(* CODESYS project 07052026.export

Project tree, tasks and I/O mapping:
  Device : ctrlX CORE ARM64, Bosch Rexroth AG, version 3.6.3.0
    application Application
      libraries: CXA_Datalayer, * (Bosch Rexroth AG); CXA_FileAsync, * (Bosch Rexroth AG); CXA_Motion, * (Bosch Rexroth AG); CXA_PLCopen, * (Bosch Rexroth AG); CXA_RobotFastManagement, 3.6.2.1 (Bosch Rexroth spa); VisuDialogs, * (System); CXA_EthercatMaster, * (Bosch Rexroth AG)
      task MainTask (cyclic, interval t#20ms, priority 30) calls PLC_PRG, prgRobotManagement, POU_GetBusState
      Robot_management_AddsOn/
        data type HomeStruct
        _CXA_RobotFastManagement_3_6_1_5/
          _00_RobotCofigurationSettings/
            global variables GVL_Robot_Config_Settings
          _01_GlobalVarConstRobotBase_3_6_1_5/
            global variables Global_Var_RobotBase
          _02_GlobalVarConstantRobotPathPlanner_3_6_1_5/
            global variables Global_Var_RobotPathPlanner
          _05_GlobalBeltVar_1_0/
            global variables GlobalBeltVar
          _06_RobotProgramExample_3_6_1_5/
            program prgRobotManagement [ST]: a00_RobotBase, a01_PathPlanner, a02_TeachIn, a03_Belt, a99_Examples
      global variables GVL
      program PLC_PRG [ST]
      program POU_GetBusState [ST]
      data type DUT
      trace Delta (task MainTask): stRobotFbk[1].arPathCoordinates[1], stRobotFbk[1].arPathCoordinates[2], stRobotFbk[1].arPathCoordinates[3], stRobotFbk[1].rPathVelocity, stRobotFbk[1].rPathAcceleration, stRobotFbk[1].rPathJerk, stKinPathBlendingStatus[1].bKinContourActive, stKinPathBlendingStatus[1].bPolySlopeActive, PLC_PRG.bCycleStart, stRobotPathPlanner[1].stRobotPoints[2].bMoveToDone, prgRobotManagement.fbRobotPathPlanner[1].fbMoveAbsolute1.I_SetPointType, prgRobotManagement.fbRobotPathPlanner[1].fbMoveAbsolute1.O_bKinMoveLinAbsError, PLC_PRG.bSetDriveOutput, prgRobotManagement.fbRobotPathPlanner[1].O_stPathPlannerFbk.usiBufferedBlock, prgRobotManagement.fbRobotPathPlanner[1].i, prgRobotManagement.fbRobotPathPlanner[1].bExMove, prgRobotManagement.fbRobotPathPlanner[1].iStep, prgRobotManagement.fbRobotPathPlanner[1].iBufferValue, prgRobotManagement.fbRobotPathPlanner[1].iBufferLimit, , prgRobotManagement.fbRobotPathPlanner[1].iCountCmdBuffered, PLC_PRG.fbIpoDelta.Position[1], PLC_PRG.fbIpoDelta.Position[2], PLC_PRG.fbIpoDelta.Position[3], prgRobotManagement.tCycle, PLC_PRG.bEnableCiclo, PLC_PRG.rRot, PLC_PRG.rRadius
      trace Scara (task MainTask): stRobotFbk[2].arPathCoordinates[1], stRobotFbk[2].arPathCoordinates[2], stRobotFbk[2].arPathCoordinates[6], stRobotFbk[2].rPathVelocity, stRobotFbk[2].rPathAcceleration, stRobotFbk[2].rPathJerk, stKinPathBlendingStatus[2].bKinContourActive, stKinPathBlendingStatus[2].bPolySlopeActive, PLC_PRG.bCycleStart, stRobotPathPlanner[1].stRobotPoints[2].bMoveToDone, prgRobotManagement.fbRobotPathPlanner[2].fbMoveAbsolute1.I_SetPointType, prgRobotManagement.fbRobotPathPlanner[2].fbMoveAbsolute1.O_bKinMoveLinAbsError, PLC_PRG.bSetDriveOutput, prgRobotManagement.fbRobotPathPlanner[2].O_stPathPlannerFbk.usiBufferedBlock, prgRobotManagement.fbRobotPathPlanner[2].i, prgRobotManagement.fbRobotPathPlanner[2].bExMove, prgRobotManagement.fbRobotPathPlanner[2].iStep, prgRobotManagement.fbRobotPathPlanner[2].iBufferValue, prgRobotManagement.fbRobotPathPlanner[1].iBufferLimit, , prgRobotManagement.fbRobotPathPlanner[2].iCountCmdBuffered, PLC_PRG.fbIpoDelta.Position[1], PLC_PRG.fbIpoDelta.Position[2], PLC_PRG.fbIpoDelta.Position[3], prgRobotManagement.tCycle, PLC_PRG.bEnableCiclo, PLC_PRG.rRot, PLC_PRG.rRadius
      visualisation Visualization
    Realtime_Data : DataLayer, Bosch Rexroth AG, version 3.6.2.0
  text list GlobalTextList
*)

// Device/Application/DUT
{attribute 'qualified_only'}
{attribute 'strict'}
TYPE DUT :
(
	enum_member := 0
);
END_TYPE

// Device/Application/Robot_management_AddsOn/HomeStruct
TYPE HomeStruct :
STRUCT
    FsSdoSetUp_u : UINT;
	SlaveAddress : UINT;
	WorkingMode : UINT;
    FsHoming : UINT;
    OuterAngle : REAL;
	OffesetInnerAngle_w : DINT;
	OffesetInnerAngle_r : DINT;
	HomeOffsetDone : BOOL;
	FeedConstant_w : ULINT;
	GearRatio_sub1_w : ULINT;
	GearRatio_sub2_w : ULINT;
	FeedConstant_r : ULINT;
	GearRatio_sub1_r : ULINT;
	GearRatio_sub2_r : ULINT;
	GearRatioConstant : REAL;
END_STRUCT
END_TYPE

// Device/Application/GVL
//{attribute 'qualified_only'}

VAR_GLOBAL
	//st values
	IN_OP_NO_HOMING   : UINT   			   := 0;
	FROM_OP_PREOP_HOME_NOT_DONE   : UINT   := 1;
	HOMING_DONE   : UINT   				   := 2;
	FROM_PREOP_OP_HOME_DONE   : UINT       := 3;

	HOMING_MODE : UINT := 0;
	FEED_CONSTANT : UINT := 1;
	GEAR_RATIO_SUB1 : UINT := 2;
	GEAR_RATIO_SUB2 : UINT := 3;
	METH_AND_ANGLE : UINT := 4;
	WRITE_OFFSET : UINT := 5;

	re_offset_input_angle : REAL := 0;
	ArrayCounter : UINT := 0;
	
    ElacArrayHoming : ARRAY[0..1] OF HomeStruct := [
        (
            FsSdoSetUp_u := 0,
            SlaveAddress := 1001,
			WorkingMode := 0, 
            FsHoming := 0,
            OuterAngle := 700000,
            OffesetInnerAngle_w := 700000,
			OffesetInnerAngle_r := 0,
			HomeOffsetDone := FALSE,
			FeedConstant_w := 7000,
			GearRatio_sub1_w := 1,
			GearRatio_sub2_w := 1,
			FeedConstant_r := 0,
			GearRatio_sub1_r := 0,
			GearRatio_sub2_r := 0,
			GearRatioConstant := -100
        ),
        (
            FsSdoSetUp_u := 0,
            SlaveAddress := 1002,
			WorkingMode := 0, 
            FsHoming := 0,
            OuterAngle := 700000,
            OffesetInnerAngle_w := 700000,
			OffesetInnerAngle_r := 0,
			HomeOffsetDone := FALSE,
			FeedConstant_w := 7000,
			GearRatio_sub1_w := 1,
			GearRatio_sub2_w := 1,
			FeedConstant_r := 0,
			GearRatio_sub1_r := 0,
			GearRatio_sub2_r := 0,
			GearRatioConstant := -100
        )
    ];

END_VAR

// Device/Application/Robot_management_AddsOn/_CXA_RobotFastManagement_3_6_1_5/_00_RobotCofigurationSettings/GVL_Robot_Config_Settings
	///#############################################################################################
	///  #############################################################################################
	///
	///   General Header
	///  ---------------------------------------------------------------------------------------------
	///   Shortdescription       :  
	///   Version                : 1.0.0.<br>
	///   Name                   : GT DCIT/STS<br>
	///   Date                   : 2024-10-25<br>
	///   Company                : Bosch Rexroth  S.p.A. Electric Drives and Controls<br>
	///   Target                 : CtrlX Core V.2.6.4 <br>
	///   Functional description : Define here the robots and robots Axis names
	///   Handling specials      : 
	///								* global var arRobotKinConfig name must not be changed.
	///							    * axis definition global var arRobot..n..AxisConfig name could be changed
	///								  but thenew name must be update in global var arRobotKinConfig too. 									
	///	
	///								
	///  ---------------------------------------------------------------------------------------------
	///
	///   Additional Header
	///  ---------------------------------------------------------------------------------------------
	///   Used global variables  : 
	///
	///   Used Standard Library  : []	
	///
	///   Used Standard Function Block:	
	///      
	///   Possible error codes:	
	///
	///   Last Modified Issues: 
	///											
	///  -----------------------------------------------------------------------
	///
	///
	///  ---------------------------------------------------------------------------------------------
	///
	///  #############################################################################################
	///  ############################################################################################# 
VAR_GLOBAL
	arRobot1AxisConfig: ARRAY[1..16] OF ST_AXIS_REF := [(AxisRef := (AxisName := 'Axis_1'), AxisNo := 1, AxisConfig := enPositioningAxis, AxisType := enVirtualAxis), 
														(AxisRef := (AxisName := 'Axis_2'), AxisNo := 2, AxisConfig := enPositioningAxis, AxisType := enVirtualAxis), 
														(AxisRef := (AxisName := 'Axis_3'), AxisNo := 3, AxisConfig := enPositioningAxis, AxisType := enVirtualAxis),
														(AxisRef := (AxisName := 'Axis_4'), AxisNo := 4, AxisConfig := enPositioningAxis, AxisType := enVirtualAxis), 
														(AxisRef := (AxisName := 'Axis_5'), AxisNo := 5, AxisConfig := enPositioningAxis, AxisType := enVirtualAxis), 
														(AxisRef := (AxisName := 'Axis_6'), AxisNo := 6, AxisConfig := enPositioningAxis, AxisType := enVirtualAxis)];
														
														
	arRobotKinConfig: ARRAY[1..16] OF ST_KIN_REF := [	(KinRef := (KinName := 'Rob_Arm_5dof'), KinNo := 1, arAxisRef := arRobot1AxisConfig )];
END_VAR

// Device/Application/Robot_management_AddsOn/_CXA_RobotFastManagement_3_6_1_5/_01_GlobalVarConstRobotBase_3_6_1_5/Global_Var_RobotBase
{attribute 'symbol' := 'readwrite'}
{attribute 'linkalways' := ''}
VAR_GLOBAL
	///#############################################################################################
	///  #############################################################################################
	///
	///   General Header
	///  ---------------------------------------------------------------------------------------------
	///   Shortdescription       :  
	///   Version                : 1.0.0.<br>
	///   Name                   : GT DCIT/STS<br>
	///   Date                   : 2024-10-25<br>
	///   Company                : Bosch Rexroth  S.p.A. Electric Drives and Controls<br>
	///   Target                 : CtrlX Core V.2.6.4 <br>
	///   Functional description :  
	///   Handling specials      : 
	///							
	///	
	///								
	///  ---------------------------------------------------------------------------------------------
	///
	///   Additional Header
	///  ---------------------------------------------------------------------------------------------
	///   Used global variables  : 
	///
	///   Used Standard Library  : []	
	///
	///   Used Standard Function Block:	
	///      
	///   Possible error codes:	
	///
	///   Last Modified Issues: 
	///											
	///  -----------------------------------------------------------------------
	///
	///
	///  ---------------------------------------------------------------------------------------------
	///
	///  #############################################################################################
	///  ############################################################################################# 
	stRobotCmd: ARRAY[1..C_usiRobotNo] OF ST_Robot_CMD;
	stRobotFbk: ARRAY[1..C_usiRobotNo] OF ST_Robot_FBK;
END_VAR

// Device/Application/Robot_management_AddsOn/_CXA_RobotFastManagement_3_6_1_5/_02_GlobalVarConstantRobotPathPlanner_3_6_1_5/Global_Var_RobotPathPlanner
///#############################################################################################
///  #############################################################################################
///
///   General Header
///  ---------------------------------------------------------------------------------------------
///   Shortdescription       : Global Variable for Robot Management
///   Version                : 1.0.0.<br>
///   Name                   : GT DCIT/STS<br>
///   Date                   : 2024-10-25<br>
///   Company                : Bosch Rexroth  S.p.A. Electric Drives and Controls<br>
///   Target                 : CtrlX Core V.3.6.0 <br>
///   Functional description : 
///   Handling specials      :    -
///   
///   Last modification	  :
/// 
///   Version               : 3.6.1.3 <br>
///   Name                  : GT DCIT/STS<br>
///   Date                  : 2025-06-16<br>
///	  Company               : Bosch Rexroth  S.p.A. Electric Drives and Controls<br>
///   Target                : CtrlX Core V.3.6.0 <br>
///	  Modified POUs			: FB_RobotPathPlannerManagement<br>
///   Description 			: Chage point managament : added global cosstant to magage system buffer max full and max empty to enable to send points  <br>
///													iBufferLimit:INT:=50; 			// Higher Points Buffer Limit<br>
///													iBufferLimitMin: INT := 20;		// Lower Points Buffer Limit<br>
///													iBufferSizeContour : INT :=15 ;  // Buffer size of the kin contour function<br>
///<br>  

///
/// ---------------------------------------------------------------------------------------------
///	
///  ---------------------------------------------------------------------------------------------
{attribute 'symbol' := 'readwrite'}
VAR_GLOBAL
	stRobotPathPlanner: ARRAY[1..C_usiRobotNo] OF ST_RobotPathPlanner;
	stPathPlannerFbk: ARRAY[1..C_usiRobotNo] OF ST_PathPlanner_FBK;
	stKinPathBlendingStatus:ARRAY[1..C_usiRobotNo] OF ST_KIN_PATH_STATUS; /// Status of the kinematic blend option and contour
END_VAR

// Device/Application/Robot_management_AddsOn/_CXA_RobotFastManagement_3_6_1_5/_05_GlobalBeltVar_1_0/GlobalBeltVar
VAR_GLOBAL
	stRobotBeltManagement: ARRAY[1..C_usiRobotNo] OF ST_BeltManagement;
END_VAR

// Device/Application/PLC_PRG
PROGRAM PLC_PRG
VAR
  fbECATCoeReadSdo : IL_ECATCoeReadSdo;
  strMasterName    : STRING := 'ethercatmaster';
  boExecute        : BOOL   := FALSE;
  uiEthercatAddr   : UINT   := 1001;
  wIndex           : WORD   :=16#6061; // Identity Object
  bySubIndex       : BYTE   := 0;       // Vendor ID
  udiVendorId      : UDINT;
	bstartread: BOOL;
	// Example A : write 1 Byte value
  fbECATCoeWriteSdo : IL_ECATCoeWriteSdo;
  strMasterNameW     : STRING := 'ethercatmaster';
  uiEthercatAddrW    : UINT := 1001;
  wIndexW            : WORD := 16#6060;  // device specific Index/SubIndex
  bySubIndexW        : BYTE := 0;        // ... which is writeable!
  byWriteValue      : BYTE := 16#06;
  bstartwrite: BOOL;
END_VAR

fbECATCoeWriteSdo.Execute      := bstartwrite;
fbECATCoeWriteSdo.MasterName   := ADR(strMasterNameW);
fbECATCoeWriteSdo.SlaveAddress := 1001;
fbECATCoeWriteSdo.Index        := wIndexW;
fbECATCoeWriteSdo.SubIndex     := bySubIndexW;
fbECATCoeWriteSdo.ValueAdr     := ADR(byWriteValue);
fbECATCoeWriteSdo.SizeOfValue  := SIZEOF(byWriteValue);
fbECATCoeWriteSdo();

IF TRUE = fbECATCoeWriteSdo.Done THEN
  ; // FB finished . byWriteValue was written to slave.
END_IF
IF TRUE = fbECATCoeWriteSdo.Error THEN
  ; // Error handling
END_IF

// Example A : read Vendor ID
fbECATCoeReadSdo.Execute      := bstartread;
fbECATCoeReadSdo.MasterName   := ADR(strMasterName);
fbECATCoeReadSdo.SlaveAddress := 1001;
fbECATCoeReadSdo.Index        := wIndex;
fbECATCoeReadSdo.SubIndex     := bySubIndex;
fbECATCoeReadSdo.ValueAdr     := ADR(udiVendorId);
fbECATCoeReadSdo.SizeOfValue  := SIZEOF(udiVendorId);
fbECATCoeReadSdo();
IF TRUE = fbECATCoeReadSdo.Done THEN
  ; // FB finished . Vendor ID is in udiVendorId.
END_IF
IF TRUE = fbECATCoeReadSdo.Error THEN
  ; // Error handling
END_IF

END_PROGRAM

// Device/Application/Robot_management_AddsOn/_CXA_RobotFastManagement_3_6_1_5/_06_RobotProgramExample_3_6_1_5/prgRobotManagement
///#############################################################################################
///  #############################################################################################
///
///   General Header
///  ---------------------------------------------------------------------------------------------
///   Shortdescription       : Program call of the robot management functions block example
///   Version                : 1.0.0.<br>
///   Name                   : GT DCIT/STS<br>
///   Date                   : 2024-10-25<br>
///   Company                : Bosch Rexroth  S.p.A. Electric Drives and Controls<br>
///   Target                 : CtrlX Core V.2.6.4 <br>
///   Functional description :  
///   Handling specials      : 
///	
///								
///  ---------------------------------------------------------------------------------------------
///
///   Additional Header
///  ---------------------------------------------------------------------------------------------
///   Used global variables  : 
///
///   Used Standard Library  : 
///
///   Used Standard Function Block:	
///	
///   Possible error codes:	
///
///   Last Modified Issues: 
///	   	
///   		Version		: 14.22.1
///   		Name   		: GT DCIT/SAE1-IT
///   		Date   		: 2018-06-02				
///		Description	: a99_Example : Added Orientation axis position copy in circular end destination point	
///		
///  		Version		: 14.22.7.1
///   		Name   		: GT DCIT/SAE1-IT
///   		Date   		: 2021-05-18				
///		Description	: a99_Example : Changed palletization management example	
///  -----------------------------------------------------------------------
///
///
///  ---------------------------------------------------------------------------------------------
///
///  #############################################################################################
///  ############################################################################################# 
PROGRAM prgRobotManagement
VAR

/// Base
	stKinRef: AXES_GROUP_REF;
	fbRobotBase: ARRAY[1..C_usiRobotNo] OF FB_RobotBase_CtrlX;
	/// Path Planner
	fbRobotPathPlanner: ARRAY[1..C_usiRobotNo] OF FB_RobotPathPlanner;
	fbTeachInPoints: ARRAY[1..C_usiRobotNo] OF FB_TeachIn;
	fbRecipeManagement: ARRAY[1..C_usiRobotNo] OF FB_RecipeManager;
	fbRecipeManagementAddData: ARRAY[1..C_usiRobotNo] OF FB_RecipeManager;
	/// bypass	fbBeltManagement: ARRAY[1..C_usiRobotNo] OF FB_BeltManagement;

/// bypass	fbRecipeBeltManagement: ARRAY[1..C_usiRobotNo] OF FB_RecipeManager;
	usiRobot: USINT;
	
/// Example AuxPoint calculation move circular
	bEnableCalcAuxCircPoint: BOOL;
	stOriginPoint: ARRAY[1..16] OF LREAL;
	stDestPoint: ARRAY[1..16] OF LREAL;
	stAuxPoint: ARRAY[1..16] OF LREAL;
	bNegQuadrant: BOOL;
	
/// Example copy points inside the point table to palletize
	bTrxPoint: BOOL;
	bUpdatePlaceDone: BOOL;
	iPlace: INT;
	iPlaceMax: INT := 2;
	bPalletizeDone: BOOL;

///	Example update belt tracking points 
	bEnableExampleBeltTracking: BOOL;
	bDesynchAfterPick: BOOL;
	bDesynchAfterPlace: BOOL;
	bEnableExampleMOveJumpBeltSync: BOOL;
	fbTeachInNew: FB_TeachIn;
	strRecipeAddData: STRING(255);
	bRecipeAddDataCommandDone: BOOL;
	bRecipeCommandDone: BOOL;

//  Start a points sequence without Enable inteblocks with PolySlope or Path Smotth Slope
	fbKinSeqStart: FB_KinPathSmoothAutoSeq;
	bEnableKinSeqStart: BOOL;
	iStartPoint: INT := 2;
	iEndPoint: INT:=6;
	iRepeatCycles: INT;
	fbPolySlopeSeq: FB_KinPathPolyContAutoSeq;
	bEnableKinSeqStartPolySlope:BOOL;

//Active and manage " bSetContinousContourDisableWaitDone" using switch on path at pick done and place done
	rSwitchDistance: REAL := 20;
	rApproxWindow: REAL := 2;
	bPickDone: BOOL;
	bPlaceDone: BOOL;
	tEndTask: LTIME;
	tCycle: LTIME;
	tStartTask: LTIME;

// #############  Belt Tracking ###############
	stBeltValueData: CXA_Motion.ML_AxsGetBeltValueData;
	stTrackingBelt1: CXA_Motion.ML_KinBeltSyncPData;
	bStartBeltTracking: BOOL;
	bTrackingActiveBelt1: BOOL;
	bStopBeltTracking: BOOL;
	rTrackingPosBelt1: LREAL;
	fbReadBeltSynStatus: DL_ReadNode;
	bExReadBeltSynStatus: BOOL;
	outValueReadBeltSynStatus: STRING;
	bSetBeltTrackingPickDone: BOOL;
	bEnableBeltTracking:BOOL;

// ########## Belt Axis Commands Example #########################
// ###################  Belt Axis #############################
	
	fbPowerOnBeltAxis1: MC_Power;
	fbMoveVelBeltAxis1: MC_MoveVelocity;
	fbStopBeltAxis1: MC_Stop;
	bEnPowerBeltAxis1: BOOL;
	stBeltAxis1: AXIS_REF;
	bExMoveVelBeltaAxis1: BOOL;
	rVelBeltAxis1: LREAL := 2000;
	rAccBeltAxis1: LREAL := 10000;
	bStopBeltAxis1: BOOL;
	fbReadActualPosBelt1: MC_ReadActualPosition;
	
	fbPowerOnBeltAxis2: MC_Power;
	fbMoveVelBeltAxis2: MC_MoveVelocity;
	fbStopBeltAxis2: MC_Stop;
	bEnPowerBeltAxis2: BOOL;
	stBeltAxis2: AXIS_REF;
	bExMoveVelBeltaAxis2: BOOL;
	rVelBeltAxis2: LREAL := 2000;
	rAccBeltAxis2: LREAL := 10000;
	bStopBeltAxis2: BOOL;
	fbReadActualPosBelt2: MC_ReadActualPosition;
	
	
END_VAR

tStartTask := LTIME();
// Robot management
FOR usiRobot := 1 TO C_usiRobotNo DO
	a00_RobotBase();
	a01_PathPlanner();
	a02_TeachIn();	
	// a03_Belt();
	// a99_Examples();
END_FOR
tEndTask := LTIME();
tCycle:=tEndTask-tStartTask;

ACTION a00_RobotBase:

fbRobotBase[usiRobot](
			I_bEnable:= stRobotCmd[usiRobot].bEnable, 
			I_KinRef:= arRobotKinConfig[usiRobot], 
			I_stRobotCmd:= stRobotCmd[usiRobot], 
			I_stRobot1AxisConfig:= arRobotKinConfig[usiRobot].arAxisRef,
			O_stRobotFbk=> stRobotFbk[usiRobot],
			O_bErrorFB=>,
			O_uiErrorCodeFB=>,
			O_strErrorIdent=>);
END_ACTION

ACTION a01_PathPlanner:


fbRobotPathPlanner[usiRobot](
	I_bEnable:= stRobotPathPlanner[usiRobot].stPathPlannerCmd.bRunPathPlanner, 
	I_HoldCycle:=stRobotPathPlanner[usiRobot].stPathPlannerCmd.bHoldCycle,
	I_usiStepsNo:=stRobotPathPlanner[usiRobot].stPathPlannerCmd.iStepNo, 
	I_stKinRef:= arRobotKinConfig[usiRobot] , 
	I_stPathPlannerCmd:=stRobotPathPlanner[usiRobot].stPathPlannerCmd,
	I_stMoveCircAddData:=stRobotPathPlanner[usiRobot].stMoveCircAddData,
	I_stRobotFbk:=stRobotFbk[usiRobot] , 
	IO_stRobotPoints:= stRobotPathPlanner[usiRobot].stRobotPoints, 
	IO_stKinPathStatus:=stKinPathBlendingStatus[usiRobot],
	O_stPathPlannerFbk=> stPathPlannerFbk[usiRobot], 
	O_Error=> , 
	O_ErrorID=> , 
	O_ErrorIdent=> );
END_ACTION

ACTION a02_TeachIn:

			
fbTeachInPoints[usiRobot](
			I_bEnable:= stRobotCmd[usiRobot].bEnable, 
			I_KinRef:= stKinRef, 
			I_stRobotFbk:=stRobotFbk[usiRobot],
			I_bExTeachIn:=stRobotPathPlanner[usiRobot].stTeachInPoints.bExTeachIn ,  
			I_bExTeachInAuxCirc:= stRobotPathPlanner[usiRobot].stTeachInPoints.bExTeachInAuxCirc, 
			I_usiSetPointNo:= stRobotPathPlanner[usiRobot].stTeachInPoints.usiSetPointNo, 
			IO_usiPointNo:= stRobotPathPlanner[usiRobot].stTeachInPoints.usiTeachInPoint, 
			IO_stRobotPoints:= stRobotPathPlanner[usiRobot].stRobotPoints, 
			O_bTeachInDone=> stRobotPathPlanner[usiRobot].stTeachInPoints.bTeachInDone);
			
			
fbRecipeManagement[usiRobot]( 
			I_bExecute:= stRobotPathPlanner[usiRobot].stTeachInPoints.bExRecipeCommand, 
			I_strSourceFileName:= stRobotPathPlanner[usiRobot].stTeachInPoints.strCopyRecipeFile, 
			I_strDestFileName:= stRobotPathPlanner[usiRobot].stTeachInPoints.strRecipeFile, 
			I_dwPtrToArray:= ADR(stRobotPathPlanner[usiRobot].stRobotPoints) , 
			I_dwArraySize:= SIZEOF (stRobotPathPlanner[usiRobot].stRobotPoints),
			I_enCommand:= stRobotPathPlanner[usiRobot].stTeachInPoints.enRecipeCommand, 
			O_bActive=> , 
			O_bDone=>bRecipeCommandDone , 
			O_bCommandAborted=> , 
			O_bError=> , 
			O_wErrorId=> , 
			O_strErrorIdent=> );			
								
strRecipeAddData := CONCAT(STR1:= stRobotPathPlanner[usiRobot].stTeachInPoints.strRecipeFile , STR2:='_AddData' );						
fbRecipeManagementAddData[usiRobot]( 
			I_bExecute:= stRobotPathPlanner[usiRobot].stTeachInPoints.bExRecipeCommand, 
			I_strSourceFileName:= stRobotPathPlanner[usiRobot].stTeachInPoints.strCopyRecipeFile, 
			I_strDestFileName:= strRecipeAddData, 
			I_dwPtrToArray:= ADR(stRobotPathPlanner[usiRobot].stMoveCircAddData) , 
			I_dwArraySize:= SIZEOF (stRobotPathPlanner[usiRobot].stMoveCircAddData),
			I_enCommand:= stRobotPathPlanner[usiRobot].stTeachInPoints.enRecipeCommand, 
			O_bActive=> , 
			O_bDone=> bRecipeAddDataCommandDone, 
			O_bCommandAborted=> , 
			O_bError=> , 
			O_wErrorId=> , 
			O_strErrorIdent=> );		
		
stRobotPathPlanner[usiRobot].stTeachInPoints.bRecipeCommandDone:=	bRecipeAddDataCommandDone AND bRecipeCommandDone;
END_ACTION

ACTION a03_Belt:
(* bypass
fbBeltManagement[usiRobot](
	I_bEnable:=stRobotBeltManagement[usiRobot].bEnable, 
	I_KinRef:= stKinRef, 
	I_stRobotCmd:= stRobotCmd[usiRobot],  
	I_stRobotFbk:= stRobotFbk[usiRobot], 
	I_stRobotBeltManagement:= stRobotBeltManagement[usiRobot], 
	O_BeltConfigDone:= , 
	O_bErrorFB:= , 
	O_uiErrorCodeFB:= , 
	O_strErrorIdent:= );
	
	
fbRecipeBeltManagement[usiRobot]( 
			I_bExecute:= stRobotBeltManagement[usiRobot].bExRecipeCommand, 
			I_strSourceFileName:= stRobotBeltManagement[usiRobot].strCopyRecipeFile, 
			I_strDestFileName:= stRobotBeltManagement[usiRobot].strRecipeFile, 
			I_dwPtrToArray:= ADR ( stRobotBeltManagement[usiRobot].arBeltConfig), 
			I_dwArraySize:= SIZEOF ( stRobotBeltManagement[usiRobot].arBeltConfig),
			I_enCommand:= stRobotBeltManagement[usiRobot].enRecipeCommand, 
			O_bActive=> , 
			O_bDone=> stRobotBeltManagement[usiRobot].bRecipeCommandDone, 
			O_bCommandAborted=> , 
			O_bError=> , 
			O_wErrorId=> , 
			O_strErrorIdent=> );		
	
	*)
END_ACTION

ACTION a99_Examples:

// ******************************** Example calculate aux circular point ******************************************
IF bEnableCalcAuxCircPoint THEN

	// Calculate Circular AuxPoint Example
	FN_AuxCirclePoint(	I_arPointOrigin:= stOriginPoint  , 
						I_arPointDestination:=  stDestPoint, 
						I_bNegQuadrant:= bNegQuadrant, 
						I_enRoundCoord:= enX_Y, 
						I_bOrientAxisCoord:=0,
						O_arAuxPoint=>  stAuxPoint);
						
	// Calculate Circular AuxPoint Example round block 2-3 program 
	FN_AuxCirclePoint(	I_arPointOrigin:= stRobotPathPlanner[1].stRobotPoints[2].arPos  , 
						I_arPointDestination:= stRobotPathPlanner[1].stRobotPoints[3].arPos, 
						I_bNegQuadrant:= bNegQuadrant, 
						I_enRoundCoord:= enX_Y, 
						I_bOrientAxisCoord:=0,
						O_arAuxPoint=> stRobotPathPlanner[1].stRobotPoints[3].arAuxPos);
					
END_IF

// ********************************* Start a points sequence without Enable inteblocks with PolySlope or Path Smotth Slope ****************************************************

fbKinSeqStart(
	I_bEnable:= bEnableKinSeqStart, 
	I_uiInitPointNo:= iStartPoint, 
	I_uiEndPointNo:= iEndPoint, 
	I_stKinRef:=arRobotKinConfig[1],  
	I_iRepeatCycles:= iRepeatCycles, 
	O_bActive=> , 
	O_bInputParametersError=> , 
	O_bSigleCycleBufferedDone=> , 
	O_bCompleteCyclesBufferedDone=> , 
	O_uiNoOfBufferedCycles=> , 
	IO_stRobotPoints:= stRobotPathPlanner[1].stRobotPoints);
	
fbPolySlopeSeq(
	I_bEnable:=bEnableKinSeqStartPolySlope , 
	I_uiInitPointNo:= iStartPoint, 
	I_uiEndPointNo:= iEndPoint, 
	I_stKinRef:=arRobotKinConfig[1],  
	I_iRepeatCycles:= iRepeatCycles, 
	O_bActive=> , 
	O_bInputParametersError=> , 
	O_bSigleCycleBufferedDone=> , 
	O_bCompleteCyclesBufferedDone=> , 
	O_uiNoOfBufferedCycles=> , 
	IO_stRobotPoints:= stRobotPathPlanner[1].stRobotPoints);


// ******************************** Ottimization of path calculation " bSetAlwaysKinCountour" using switch on path at pick done and place done ************************************** 

FN_SwitchOnPath(
	Enable:= stRobotPathPlanner[1].stPathPlannerCmd.bRunPathPlanner, 
	Target:= stRobotPathPlanner[1].stRobotPoints[3].arPos, // Pick position
	FeedBack:=stRobotFbk[1].arPathCoordinates, 
	SwitchDist:= rSwitchDistance, 
	ApproxWindow:= rApproxWindow, 
	InOperation=> , 
	InRange=> bPickDone, 
	Error=> );

	
FN_SwitchOnPath(
	Enable:= stRobotPathPlanner[1].stPathPlannerCmd.bRunPathPlanner, 
	Target:= stRobotPathPlanner[1].stRobotPoints[6].arPos, // place position
	FeedBack:=stRobotFbk[1].arPathCoordinates, 
	SwitchDist:= rSwitchDistance, 
	ApproxWindow:= rApproxWindow, 
	InOperation=> , 
	InRange=> bPlaceDone, 
	Error=> );
	
	stRobotPathPlanner[1].stRobotPoints[4].bEnableCondition:=bPickDone;
	
	stRobotPathPlanner[1].stRobotPoints[7].bEnableCondition:=bPlaceDone;
	
	IF stPathPlannerFbk[1].usiBufferedBlock >=2 THEN 
		stRobotPathPlanner[1].stPathPlannerCmd.bSetAlwaysKinContour:=TRUE;	
	ELSE
		stRobotPathPlanner[1].stPathPlannerCmd.bSetAlwaysKinContour:=FALSE;
	END_IF	

					
// ******************************** Example copy points inside the point table ( Palletizer ) **************************************
IF bTrxPoint THEN
	
	IF stRobotPathPlanner[1].stPathPlannerCmd.bRunPathPlanner = FALSE THEN
		bUpdatePlaceDone:=FALSE;
		iPlace:=0;
	END_IF

	(* Copy placement points layers on pallet *)
	IF stPathPlannerFbk[1].usiBufferedBlock = 3  THEN
		bUpdatePlaceDone:=FALSE;
		CASE iPlace OF
		
		0:
			// Copy place points product 1 to place points run
			prgRobotManagement.fbRobotPathPlanner[1].mCopyBlock(101,5);
			prgRobotManagement.fbRobotPathPlanner[1].mCopyBlock(102,6);
			prgRobotManagement.fbRobotPathPlanner[1].mCopyBlock(103,7);
	
			
		1:
			// Copy place points product 2 to place points run
			prgRobotManagement.fbRobotPathPlanner[1].mCopyBlock(111,5);
			prgRobotManagement.fbRobotPathPlanner[1].mCopyBlock(112,6);
			prgRobotManagement.fbRobotPathPlanner[1].mCopyBlock(113,7);
		
		
		2:
			// Copy place points product 3 to place points run
			prgRobotManagement.fbRobotPathPlanner[1].mCopyBlock(121,5);
			prgRobotManagement.fbRobotPathPlanner[1].mCopyBlock(122,6);
			prgRobotManagement.fbRobotPathPlanner[1].mCopyBlock(123,7);
			
		3:
			// Copy place points product n to place points run
		
	
		END_CASE
	
	END_IF
	
	// Place Point Block Done
	IF stPathPlannerFbk[1].usiBufferedBlock = 6 AND   stPathPlannerFbk[1].bMoveToDone AND NOT bUpdatePlaceDone THEN
		bUpdatePlaceDone:=TRUE;
		IF iPlace < iPlaceMax  THEN
			iPlace:=iPlace +1;
		ELSE
			iPlace:=0;
			bPalletizeDone:=TRUE; 
		END_IF
	END_IF
END_IF	

// ******************************** Example belt tracking points update management ******************************************************
// Enable Example Belt Tracking Point Management
FN_SwitchOnPath(
	Enable:= stRobotPathPlanner[1].stPathPlannerCmd.bRunPathPlanner, 
	Target:= stRobotPathPlanner[1].stRobotPoints[3].arPos, // Pick position
	FeedBack:=stRobotFbk[1].arPathCoordinates, 
	SwitchDist:= rSwitchDistance, 
	ApproxWindow:= rApproxWindow, 
	InOperation=> , 
	InRange=> bPickDone, 
	Error=> );

	
FN_SwitchOnPath(
	Enable:= stRobotPathPlanner[1].stPathPlannerCmd.bRunPathPlanner, 
	Target:= stRobotPathPlanner[1].stRobotPoints[6].arPos, // place position
	FeedBack:=stRobotFbk[1].arPathCoordinates, 
	SwitchDist:= rSwitchDistance, 
	ApproxWindow:= rApproxWindow, 
	InOperation=> , 
	InRange=> bPlaceDone, 
	Error=> );
	
	IF stKinPathBlendingStatus[1].stBeltTrackingStatus.SYNCHRONIZED AND stRobotFbk[1].arPathCoordinates[3] <= stRobotPathPlanner[1].stRobotPoints[3].arPos[3] 
		OR stRobotPathPlanner[1].stRobotPoints[3].bMoveToDone THEN
		bPickDone:=TRUE;
	ELSE
		bPickDone:=FALSE;
	END_IF
	
	// Tracking Pick Points
	stBeltValueData.In.AxisName := 'Belt1';
	ML_AxsGetBeltValueRT(Data:= stBeltValueData); //read current belt value	
	rTrackingPosBelt1:= (TRUNC(stBeltValueData.Out.Position*1000)/1000);
	rTrackingPosBelt1:=rTrackingPosBelt1/1000;
	IF rTrackingPosBelt1 < 0.001 THEN
		rTrackingPosBelt1 :=0.001;
	END_IF
	
	IF (stPathPlannerFbk[1].usiBufferedBlock <2  OR ( stPathPlannerFbk[1].usiBufferedBlock >=5 AND stPathPlannerFbk[1].usiBufferedBlock <=7 ) )  
		AND stKinPathBlendingStatus[1].stBeltTrackingStatus.DESYNCHRONIZED  AND NOT bSetBeltTrackingPickDone AND bEnableBeltTracking THEN  
		
		// Up Pick Synchro down direction
		stRobotPathPlanner[1].stRobotPoints[2].arPos[9]:=rTrackingPosBelt1;
		stRobotPathPlanner[1].stRobotPoints[2].arPos[10]:=0;
		// Pick Synchro
		stRobotPathPlanner[1].stRobotPoints[3].arPos[9]:=rTrackingPosBelt1;
		stRobotPathPlanner[1].stRobotPoints[3].arPos[10]:=0;
		// Up Pick Synchro up direction
		stRobotPathPlanner[1].stRobotPoints[4].arPos[9]:=rTrackingPosBelt1;
		stRobotPathPlanner[1].stRobotPoints[4].arPos[10]:=0;
		bSetBeltTrackingPickDone:=TRUE;
	END_IF
	
	IF stKinPathBlendingStatus[1].stBeltTrackingStatus.SYNCHRONIZED  OR stKinPathBlendingStatus[1].stBeltTrackingStatus.SYNCHRONIZING 
		OR NOT stRobotPathPlanner[1].stPathPlannerCmd.bRunPathPlanner   THEN
		bSetBeltTrackingPickDone:=FALSE;
	END_IF	
	
	
	IF bEnableBeltTracking THEN
		stRobotPathPlanner[1].stRobotPoints[2].bEnableCondition:= bSetBeltTrackingPickDone  ;
		stRobotPathPlanner[1].stRobotPoints[4].bEnableCondition:=bPickDone;
		bPlaceDone:= stRobotPathPlanner[1].stRobotPoints[6].bMoveToDone;
		stRobotPathPlanner[1].stRobotPoints[7].bEnableCondition:=bPlaceDone;
	END_IF
	
	// ***************************************************** ABSOLUTE DESYNCRONIZATION ********************************************
	// Desynch if no place point available after pick 
	IF bDesynchAfterPick THEN // Missing Place po0int after pick done
		IF stPathPlannerFbk[1].usiBufferedBlock = 4 THEN
			stRobotPathPlanner[1].stRobotPoints[4].usiJumpAfter:=1; // Go to Home
			stRobotPathPlanner[1].stPathPlannerCmd.bInTouchProbeStop:=TRUE;
		END_IF
		IF stPathPlannerFbk[1].usiBufferedBlock = 1 THEN
			stRobotPathPlanner[1].stPathPlannerCmd.bInTouchProbeStop:=FALSE;
			bDesynchAfterPick:=FALSE;
			stRobotPathPlanner[1].stRobotPoints[1].usiJumpAfter:=0; // Stay in Home
		END_IF
	END_IF
	// Desynch if no pick point available after place 
	IF bDesynchAfterPlace THEN // Missing Place po0int after pick done
		IF stPathPlannerFbk[1].usiBufferedBlock = 7 THEN
			stRobotPathPlanner[1].stRobotPoints[7].usiJumpAfter:=1; // Go to Home
			stRobotPathPlanner[1].stPathPlannerCmd.bInTouchProbeStop:=TRUE;
		END_IF
		IF stPathPlannerFbk[1].usiBufferedBlock = 1 THEN
			stRobotPathPlanner[1].stPathPlannerCmd.bInTouchProbeStop:=FALSE;
			bDesynchAfterPlace:=FALSE;
			stRobotPathPlanner[1].stRobotPoints[1].usiJumpAfter:=0; // Stay in Home
		END_IF
	END_IF
	
	
// ######################################### Belt Axis Commands Example ###########################################################


stBeltAxis1.AxisName:='Belt1';

fbPowerOnBeltAxis1(
	Enable:= bEnPowerBeltAxis1, 
	Status=> , 
	Error=> , 
	ErrorID=> , 
	ErrorIdent=> , 
	Axis:=stBeltAxis1 );
	
fbMoveVelBeltAxis1(
	Execute:= bExMoveVelBeltaAxis1, 
	ContinuousUpdate:= , 
	Velocity:= rVelBeltAxis1, 
	DriveVelMode:= , 
	Acceleration:= rAccBeltAxis1, 
	Deceleration:= rAccBeltAxis1, 
	Jerk:= , 
	BufferMode:= , 
	InVelocity=> , 
	Busy=> , 
	Active=> , 
	CommandAborted=> , 
	Error=> , 
	ErrorID=> , 
	ErrorIdent=> , 
	Axis:=stBeltAxis1 );
	
fbStopBeltAxis1(
	Execute:=bStopBeltAxis1 , 
	Deceleration:= rAccBeltAxis1, 
	Jerk:= , 
	UseAH:= , 
	Done=> , 
	Active=> , 
	CommandAborted=> , 
	Error=> , 
	ErrorID=> , 
	ErrorIdent=> , 
	Axis:= stBeltAxis1);	
	
fbReadActualPosBelt1(
	Enable:= bEnPowerBeltAxis1, 
	Valid=> , 
	Active=> , 
	Error=> , 
	ErrorID=> , 
	ErrorIdent=> , 
	Position=> , 
	Axis:=stBeltAxis1 );	
	
stBeltAxis2.AxisName:='Belt2';

fbPowerOnBeltAxis2(
	Enable:= bEnPowerBeltAxis2, 
	Status=> , 
	Error=> , 
	ErrorID=> , 
	ErrorIdent=> , 
	Axis:=stBeltAxis2 );
	
fbMoveVelBeltAxis2(
	Execute:= bExMoveVelBeltaAxis2, 
	ContinuousUpdate:= , 
	Velocity:= rVelBeltAxis2, 
	DriveVelMode:= , 
	Acceleration:= rAccBeltAxis2, 
	Deceleration:= rAccBeltAxis2, 
	Jerk:= , 
	BufferMode:= , 
	InVelocity=> , 
	Busy=> , 
	Active=> , 
	CommandAborted=> , 
	Error=> , 
	ErrorID=> , 
	ErrorIdent=> , 
	Axis:=stBeltAxis2 );
	
fbStopBeltAxis2(
	Execute:=bStopBeltAxis2, 
	Deceleration:= rAccBeltAxis2, 
	Jerk:= , 
	UseAH:= , 
	Done=> , 
	Active=> , 
	CommandAborted=> , 
	Error=> , 
	ErrorID=> , 
	ErrorIdent=> , 
	Axis:= stBeltAxis2);	
	
fbReadActualPosBelt2(
	Enable:= TRUE, 
	Valid=> , 
	Active=> , 
	Error=> , 
	ErrorID=> , 
	ErrorIdent=> , 
	Position=> , 
	Axis:=stBeltAxis2 );		
	
(* bypass	
	// ***************************************************** MOVE JUMP Belt Synch ***********************************************************
IF bEnableExampleMOveJumpBeltSync THEN 
		
	// ******************************* NOTE ON MOVEJUMP SYNCH TO BELT ***************************************
	(*
		If the following Move Jump point is not in the belt area the robot stay synhcronizaed to the belt down in the previous reaced point.
		To avoid this is necessary to program a Move Jump Up ( home ) point to desynchronize from the previous belt when the point on the next belt is not in the belt area
		( see point 14 and point 17 in the recipe file "delta1_reldesync_moveJump" used in the following example )
	*)
	// ************************************* END NOTE *******************************************************

	// Tracking Points from home to pick
	IF stPathPlannerFbk[1].usiBufferedBlock <Point2  THEN 
		stRobotPathPlanner[1].stRobotPoints[Point12].arPos[1]:=stRobotBeltManagement[1].arBeltConfig[1].rXposBelt;
		stRobotPathPlanner[1].stRobotPoints[Point12].arPos[5]:=KinData[1].arPositionOriginalCoord_i[5];
		stRobotPathPlanner[1].stRobotPoints[Point12].arPos[6]:=0;
	END_IF
	
	// Tracking Points from pick to place
	IF  stPathPlannerFbk[1].usiBufferedBlock <Point2 OR stPathPlannerFbk[1].usiBufferedBlock = Point12  OR stPathPlannerFbk[1].usiBufferedBlock = Point13  OR stPathPlannerFbk[1].usiBufferedBlock = Point14 THEN 
		stRobotPathPlanner[1].stRobotPoints[Point16].arPos[1]:=stRobotBeltManagement[1].arBeltConfig[2].rXposBelt;
		stRobotPathPlanner[1].stRobotPoints[Point16].arPos[5]:=0;
		stRobotPathPlanner[1].stRobotPoints[Point16].arPos[6]:=KinData[1].arPositionOriginalCoord_i[6];
	
	END_IF
	
		// Tracking Points from place to pick
	IF stPathPlannerFbk[1].usiBufferedBlock = Point16 OR stPathPlannerFbk[1].usiBufferedBlock = Point17  THEN 
		stRobotPathPlanner[1].stRobotPoints[Point13].arPos[1]:=stRobotBeltManagement[1].arBeltConfig[1].rXposBelt;
		stRobotPathPlanner[1].stRobotPoints[Point13].arPos[5]:=KinData[1].arPositionOriginalCoord_i[5];
		stRobotPathPlanner[1].stRobotPoints[Point13].arPos[6]:=0;
	END_IF

END_IF
*)
END_ACTION

END_PROGRAM

// Device/Application/POU_GetBusState
PROGRAM POU_GetBusState
VAR
  fbECATMasterSetBusState: IL_ECATMasterSetBusState;
  udiSdoRead      : UDINT;
  fbECATMasterGetBusState: IL_ECATMasterGetBusState;
  eActBusState :           IL_ECAT_STATE;
  fbECATCoeReadSdo : IL_ECATCoeReadSdo;
  fbECATCoeWriteSdo : IL_ECATCoeWriteSdo;
  wIndex           : WORD   :=16#6061; // Identity Object
  bySubIndex       : BYTE   := 0;       // Vendor ID
  wIndexW            : WORD := 16#6060;  // device specific Index/SubIndex
  bySubIndexW        : BYTE := 0;        // ... which is writeable!
  byWriteValue      : BYTE := 16#06;
END_VAR


VAR CONSTANT
  FEED_COSTANT : UINT := 6000;
  GEAR_RATIO   : INT  := -100;
  ROUND_ANGLE  : UINT := 360;
  strMasterName:           STRING := 'ethercatmaster';
  HOMING_MODE_6061 : UINT := 6;
END_VAR

fbECATMasterSetBusState.Execute     := FALSE;
fbECATMasterSetBusState.MasterName  := ADR(strMasterName);
fbECATMasterGetBusState.MasterName := ADR(strMasterName);






fbECATMasterGetBusState();

// IF FALSE = fbECATMasterSetBusState.Done AND 
//    TRUE = fbECATMasterGetBusState.Done AND 
//    fbECATMasterGetBusState.ActBusState = IL_ECAT_STATE.ECAT_STATE_OP AND  
//    ElacArrayHoming[ArrayCounter].FsHoming = IN_OP_NO_HOMING THEN
//    
//   fbECATMasterSetBusState.Execute := TRUE;
//   fbECATMasterSetBusState.NewBusState := IL_ECAT_STATE.ECAT_STATE_PREOP;
//   eActBusState := fbECATMasterGetBusState.ActBusState;
// END_IF

IF  ElacArrayHoming[0].FsHoming = FROM_PREOP_OP_HOME_DONE
AND ElacArrayHoming[1].FsHoming = FROM_PREOP_OP_HOME_DONE THEN
	fbECATMasterSetBusState.Execute := TRUE;
	fbECATMasterSetBusState.NewBusState := IL_ECAT_STATE.ECAT_STATE_OP;
END_IF

//IF TRUE = fbECATMasterSetBusState.Done AND ElacArrayHoming[ArrayCounter].FsHoming <> FROM_PREOP_OP_HOME_DONE THEN
IF fbECATMasterGetBusState.ActBusState = IL_ECAT_STATE.ECAT_STATE_PREOP THEN	
	fbECATCoeReadSdo.SlaveAddress := ElacArrayHoming[ArrayCounter].SlaveAddress;
	fbECATCoeWriteSdo.SlaveAddress := ElacArrayHoming[ArrayCounter].SlaveAddress;
	fbECATCoeWriteSdo.MasterName   := ADR(strMasterName);
	fbECATCoeReadSdo.MasterName   := ADR(strMasterName);
	
	IF ElacArrayHoming[ArrayCounter].FsSdoSetUp_u = HOMING_MODE THEN
		wIndex       := 16#6061; // Identity Object
		bySubIndex          := 0;       // Vendor ID
		wIndexW           := 16#6060;  // device specific Index/SubIndex
		bySubIndexW        := 0;        // ... which is writeable!
		byWriteValue     := 16#06;

		fbECATCoeWriteSdo.Execute      := TRUE;
		fbECATCoeWriteSdo.Index        := wIndexW;
		fbECATCoeWriteSdo.SubIndex     := bySubIndexW;
		fbECATCoeWriteSdo.ValueAdr     := ADR(byWriteValue);
		fbECATCoeWriteSdo.SizeOfValue  := SIZEOF(byWriteValue);
		fbECATCoeReadSdo.Execute      := TRUE;
		fbECATCoeReadSdo.Index        := wIndex;
		fbECATCoeReadSdo.SubIndex     := bySubIndex;
		fbECATCoeReadSdo.ValueAdr     := ADR(ElacArrayHoming[ArrayCounter].WorkingMode);
		fbECATCoeReadSdo.SizeOfValue  := SIZEOF(ElacArrayHoming[ArrayCounter].WorkingMode);
	END_IF
	
	IF  ElacArrayHoming[ArrayCounter].FsSdoSetUp_u = METH_AND_ANGLE THEN 
		wIndexW := 16#6098;
		byWriteValue := 37; // setting homing method 37
		wIndex := 16#201F;
		bySubIndexW := 0;
		bySubIndex := 0;
		
		fbECATCoeWriteSdo.Execute      := TRUE;
		fbECATCoeWriteSdo.Index        := wIndexW;
		fbECATCoeWriteSdo.SubIndex     := bySubIndexW;
		fbECATCoeWriteSdo.ValueAdr     := ADR(byWriteValue);
		fbECATCoeWriteSdo.SizeOfValue  := SIZEOF(byWriteValue);
		fbECATCoeReadSdo.Execute      := TRUE;
		fbECATCoeReadSdo.Index        := wIndex;
		fbECATCoeReadSdo.SubIndex     := bySubIndex;
		fbECATCoeReadSdo.ValueAdr     := ADR(ElacArrayHoming[ArrayCounter].OuterAngle);
		fbECATCoeReadSdo.SizeOfValue  := SIZEOF(ElacArrayHoming[ArrayCounter].OuterAngle);
		//re_offset_input_angle := ((ElacArrayHoming[0].OuterAngle*FEED_COSTANT*GEAR_RATIO)/(ROUND_ANGLE));
		
	END_IF
	
		IF  ElacArrayHoming[ArrayCounter].FsSdoSetUp_u = FEED_CONSTANT THEN 
		wIndexW := 16#6092; //Feed constant 
		wIndex := 16#6092; //Feed constant 
		bySubIndexW := 1;
		bySubIndex := 1;
		
		fbECATCoeWriteSdo.Execute      := TRUE;
		fbECATCoeWriteSdo.Index        := wIndexW;
		fbECATCoeWriteSdo.SubIndex     := bySubIndexW;
		fbECATCoeWriteSdo.ValueAdr     := ADR(ElacArrayHoming[ArrayCounter].FeedConstant_w);
		fbECATCoeWriteSdo.SizeOfValue  := SIZEOF(ElacArrayHoming[ArrayCounter].FeedConstant_w);
		fbECATCoeReadSdo.Execute      := TRUE;
		fbECATCoeReadSdo.Index        := wIndex;
		fbECATCoeReadSdo.SubIndex     := bySubIndex;
		fbECATCoeReadSdo.ValueAdr     := ADR(ElacArrayHoming[ArrayCounter].FeedConstant_r);
		fbECATCoeReadSdo.SizeOfValue  := SIZEOF(ElacArrayHoming[ArrayCounter].FeedConstant_r);
	END_IF
	IF  ElacArrayHoming[ArrayCounter].FsSdoSetUp_u = GEAR_RATIO_SUB1 THEN 
		wIndexW := 16#6091; //GearRatio 
		wIndex := 16#6091; //GearRatio 
		bySubIndexW := 1;
		bySubIndex := 1;
		
		fbECATCoeWriteSdo.Execute      := TRUE;
		fbECATCoeWriteSdo.Index        := wIndexW;
		fbECATCoeWriteSdo.SubIndex     := bySubIndexW;
		fbECATCoeWriteSdo.ValueAdr     := ADR(ElacArrayHoming[ArrayCounter].GearRatio_sub1_w);
		fbECATCoeWriteSdo.SizeOfValue  := SIZEOF(ElacArrayHoming[ArrayCounter].GearRatio_sub1_w);
		fbECATCoeReadSdo.Execute      := TRUE;
		fbECATCoeReadSdo.Index        := wIndex;
		fbECATCoeReadSdo.SubIndex     := bySubIndex;
		fbECATCoeReadSdo.ValueAdr     := ADR(ElacArrayHoming[ArrayCounter].GearRatio_sub1_r);
		fbECATCoeReadSdo.SizeOfValue  := SIZEOF(ElacArrayHoming[ArrayCounter].GearRatio_sub1_r);
	END_IF
		IF  ElacArrayHoming[ArrayCounter].FsSdoSetUp_u = GEAR_RATIO_SUB2 THEN 
		wIndexW := 16#6091; //GearRatio
		wIndex := 16#6091; //GearRatio
		bySubIndexW := 2;
		bySubIndex := 2;
		
		fbECATCoeWriteSdo.Execute      := TRUE;
		fbECATCoeWriteSdo.Index        := wIndexW;
		fbECATCoeWriteSdo.SubIndex     := bySubIndexW;
		fbECATCoeWriteSdo.ValueAdr     := ADR(ElacArrayHoming[ArrayCounter].GearRatio_sub2_w);
		fbECATCoeWriteSdo.SizeOfValue  := SIZEOF(ElacArrayHoming[ArrayCounter].GearRatio_sub2_w);
		fbECATCoeReadSdo.Execute      := TRUE;
		fbECATCoeReadSdo.Index        := wIndex;
		fbECATCoeReadSdo.SubIndex     := bySubIndex;
		fbECATCoeReadSdo.ValueAdr     := ADR(ElacArrayHoming[ArrayCounter].GearRatio_sub2_r);
		fbECATCoeReadSdo.SizeOfValue  := SIZEOF(ElacArrayHoming[ArrayCounter].GearRatio_sub2_r);
	END_IF
	
	IF ElacArrayHoming[ArrayCounter].FsSdoSetUp_u = WRITE_OFFSET AND ElacArrayHoming[ArrayCounter].OffesetInnerAngle_w <> 700000  THEN 
		
		wIndexW := 16#607C;
		wIndex := 16#607C;
		bySubIndexW := 0;
		bySubIndex := 0;
		
		fbECATCoeWriteSdo.Execute      := TRUE;
		fbECATCoeWriteSdo.Index        := wIndexW;
		fbECATCoeWriteSdo.SubIndex     := bySubIndexW;
		fbECATCoeWriteSdo.ValueAdr     := ADR(ElacArrayHoming[ArrayCounter].OffesetInnerAngle_w);
		fbECATCoeWriteSdo.SizeOfValue  := SIZEOF(ElacArrayHoming[ArrayCounter].OffesetInnerAngle_w);
		fbECATCoeReadSdo.Execute      := TRUE;
		fbECATCoeReadSdo.Index        := wIndex;
		fbECATCoeReadSdo.SubIndex     := bySubIndex;
		fbECATCoeReadSdo.ValueAdr     := ADR(ElacArrayHoming[ArrayCounter].OffesetInnerAngle_r);
		fbECATCoeReadSdo.SizeOfValue  := SIZEOF(ElacArrayHoming[ArrayCounter].OffesetInnerAngle_r);
	END_IF
	
	IF ElacArrayHoming[ArrayCounter].FsSdoSetUp_u = WRITE_OFFSET 
		AND ElacArrayHoming[ArrayCounter].OffesetInnerAngle_w = ElacArrayHoming[ArrayCounter].OffesetInnerAngle_r  THEN
		ElacArrayHoming[ArrayCounter].FsHoming := HOMING_DONE;
	END_IF
	
	IF ElacArrayHoming[ArrayCounter].FsSdoSetUp_u = HOMING_MODE AND ElacArrayHoming[ArrayCounter].WorkingMode = HOMING_MODE_6061 THEN 
		ElacArrayHoming[ArrayCounter].FsSdoSetUp_u := FEED_CONSTANT;		
		fbECATCoeWriteSdo.Execute      := FALSE;
		fbECATCoeReadSdo.Execute      := FALSE;
		fbECATMasterSetBusState.Execute := FALSE;
	END_IF
	
	IF ElacArrayHoming[ArrayCounter].FsHoming = HOMING_DONE THEN 
		ElacArrayHoming[ArrayCounter].FsHoming := FROM_PREOP_OP_HOME_DONE;
		fbECATCoeWriteSdo.Execute      := FALSE;
		fbECATCoeReadSdo.Execute      := FALSE;
		fbECATMasterSetBusState.Execute := FALSE;
		IF ArrayCounter < 1 THEN
			ArrayCounter := ArrayCounter +1;
		END_IF
	END_IF
	
	IF ElacArrayHoming[ArrayCounter].FsSdoSetUp_u = FEED_CONSTANT AND 
	ElacArrayHoming[ArrayCounter].FeedConstant_r = ElacArrayHoming[ArrayCounter].FeedConstant_w THEN 
		ElacArrayHoming[ArrayCounter].FsSdoSetUp_u := GEAR_RATIO_SUB1;
		fbECATCoeWriteSdo.Execute      := FALSE;
		fbECATCoeReadSdo.Execute      := FALSE;
		fbECATMasterSetBusState.Execute := FALSE;
	END_IF
	IF ElacArrayHoming[ArrayCounter].FsSdoSetUp_u = GEAR_RATIO_SUB1 AND 
	ElacArrayHoming[ArrayCounter].GearRatio_sub1_w = ElacArrayHoming[ArrayCounter].GearRatio_sub1_r THEN 
		ElacArrayHoming[ArrayCounter].FsSdoSetUp_u := GEAR_RATIO_SUB2;
		fbECATCoeWriteSdo.Execute      := FALSE;
		fbECATCoeReadSdo.Execute      := FALSE;
		fbECATMasterSetBusState.Execute := FALSE;
	END_IF
	IF ElacArrayHoming[ArrayCounter].FsSdoSetUp_u = GEAR_RATIO_SUB2 AND 
	ElacArrayHoming[ArrayCounter].GearRatio_sub2_w = ElacArrayHoming[ArrayCounter].GearRatio_sub2_r THEN 
		ElacArrayHoming[ArrayCounter].FsSdoSetUp_u := METH_AND_ANGLE;
		fbECATCoeWriteSdo.Execute      := FALSE;
		fbECATCoeReadSdo.Execute      := FALSE;
		fbECATMasterSetBusState.Execute := FALSE;
	END_IF



	
	IF ElacArrayHoming[ArrayCounter].FsSdoSetUp_u = METH_AND_ANGLE AND  ElacArrayHoming[ArrayCounter].OuterAngle <> 700000 THEN 
		ElacArrayHoming[ArrayCounter].OffesetInnerAngle_w := TO_DINT(((ElacArrayHoming[ArrayCounter].OuterAngle*TO_REAL(ElacArrayHoming[ArrayCounter].FeedConstant_w)*ElacArrayHoming[ArrayCounter].GearRatioConstant)/(ROUND_ANGLE)));
		ElacArrayHoming[ArrayCounter].FsSdoSetUp_u := WRITE_OFFSET;
		fbECATCoeWriteSdo.Execute      := FALSE;
		fbECATCoeReadSdo.Execute      := FALSE;
		fbECATMasterSetBusState.Execute := FALSE;
	END_IF
	
	IF fbECATCoeWriteSdo.Done = TRUE THEN 
		fbECATCoeWriteSdo.Execute      := FALSE;
		fbECATCoeReadSdo.Execute      := FALSE;
		fbECATMasterSetBusState.Execute := FALSE;		
	END_IF

	fbECATCoeWriteSdo();
	fbECATCoeReadSdo();
	
	IF TRUE = fbECATCoeWriteSdo.Done THEN
	  ; // FB finished . byWriteValue was written to slave.
	END_IF
	IF TRUE = fbECATCoeWriteSdo.Error THEN
	  ; // Error handling
	END_IF
	
	IF TRUE = fbECATCoeReadSdo.Done THEN
	  ; // FB finished . Vendor ID is in udiVendorId.
	END_IF
	IF TRUE = fbECATCoeReadSdo.Error THEN
	  ; // Error handling
	END_IF
END_IF

// IF ArrayCounter < 1 THEN 
// 	ArrayCounter := ArrayCounter +1;
// ELSE
// 	ArrayCounter := 0;
// END_IF

IF  FALSE = fbECATMasterSetBusState.Done THEN
	fbECATMasterGetBusState.Execute := NOT fbECATMasterGetBusState.Execute;
END_IF

fbECATMasterSetBusState();


IF TRUE = fbECATMasterSetBusState.Error THEN
  ; // error handling
END_IF

END_PROGRAM

// Device/Application/Visualization
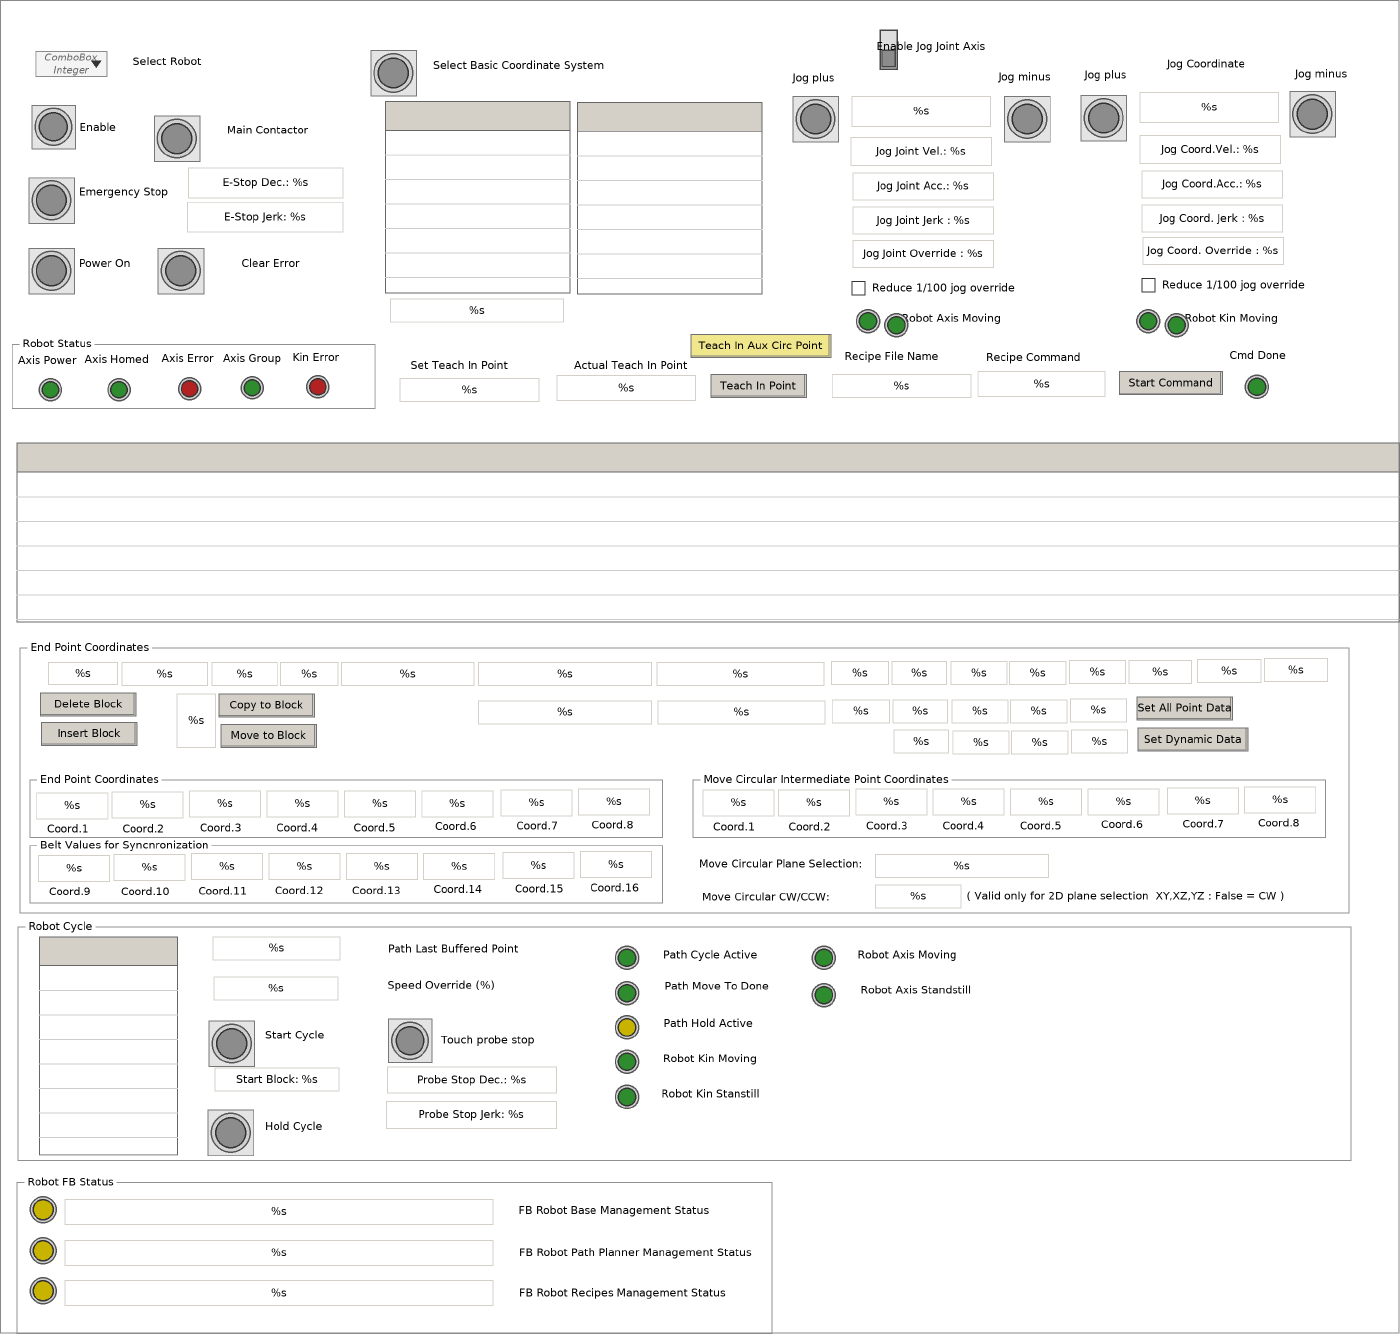
VISUALIZATION Visualization  // 1429x1362
    PushSwitch (30,107 49x45), tooltip "Enable", variable: stRobotCmd[iRobotSel].bEnable, behaviour: TOGGLE, style: Switch-PushSwitch-Gray
    PushSwitch (157,111 47x61), tooltip "Main Contactor", variable: stRobotCmd[iRobotSel].bMainContactor, behaviour: TOGGLE, style: Switch-PushSwitch-Gray
    PushSwitch (29,174 47x61), tooltip "Emergency Stop", variable: stRobotCmd[iRobotSel].bEmergencyStop, behaviour: TOGGLE, style: Switch-PushSwitch-Gray
    PushSwitch (29,246 47x61), tooltip "Power On", variable: stRobotCmd[iRobotSel].bPowerON, behaviour: TOGGLE, style: Switch-PushSwitch-Gray
    PushSwitch (809,91 47x61), tooltip "Jog Joint Plus", variable: stRobotCmd[iRobotSel].stJogJoint.bJogPos, behaviour: TAP, style: Switch-PushSwitch-Gray
    PushSwitch (1025,91 47x61), tooltip "Jog Joint Minus", variable: stRobotCmd[iRobotSel].stJogJoint.bJogNeg, behaviour: TAP, style: Switch-PushSwitch-Gray
    Textfield (869,98 142x31), "%s", text variable: stRobotCmd[iRobotSel].stJogJoint.enJogCoord
        OnMouseClick: write the text variable via Default
    PushSwitch (1103,90 47x61), tooltip "Jog Coord. Plus", variable: stRobotCmd[iRobotSel].stJogCoordinate.bJogPos, behaviour: TAP, style: Switch-PushSwitch-Gray
    PushSwitch (1316,86 47x61), tooltip "Jog Joint Minus", variable: stRobotCmd[iRobotSel].stJogCoordinate.bJogNeg, behaviour: TAP, style: Switch-PushSwitch-Gray
    Textfield (1163,94 142x31), "%s", text variable: stRobotCmd[iRobotSel].stJogCoordinate.enJogCoord
        OnMouseClick: write the text variable via Default
    Table (393,103 189x196), data array: stRobotFbk[iRobotSel].arPathCoordinates
        p3854506369: stRobotFbk[iRobotSel].arPathCoordinates[INDEX]
        p1014161805: 16 - 1 + 1
    Table (17,452 1412x183), data array: stRobotPathPlanner[iRobotSel].stRobotPoints
        p1137915858: iRowSel
        p1014161805: Robots_Constants_Settings.MaxBlocksNo - 1 + 1
        p3854506369: stRobotPathPlanner[iRobotSel].stRobotPoints[INDEX].strPointName
        p1892666644: stRobotPathPlanner[iRobotSel].stRobotPoints[INDEX].bEnableCondition
        p338671338: stRobotPathPlanner[iRobotSel].stRobotPoints[INDEX].usiJumpBefore
        p2170511999: stRobotPathPlanner[iRobotSel].stRobotPoints[INDEX].usiJumpAfter
        p3723444502: stRobotPathPlanner[iRobotSel].stRobotPoints[INDEX].enMotionType
        p1218418051: stRobotPathPlanner[iRobotSel].stRobotPoints[INDEX].enCoordSys
        p746581629: stRobotPathPlanner[iRobotSel].stRobotPoints[INDEX].enSlopeType
        p3104783080: stRobotPathPlanner[iRobotSel].stRobotPoints[INDEX].enSetMode
        p2501879983: stRobotPathPlanner[iRobotSel].stRobotPoints[INDEX].arPos
        p7306298: stRobotPathPlanner[iRobotSel].stRobotPoints[INDEX].arAuxPos
        p1933151965: stRobotPathPlanner[iRobotSel].stRobotPoints[INDEX].rVel
        p3863566920: stRobotPathPlanner[iRobotSel].stRobotPoints[INDEX].rAcc
        p2192122294: stRobotPathPlanner[iRobotSel].stRobotPoints[INDEX].rJerk
        p400160035: stRobotPathPlanner[iRobotSel].stRobotPoints[INDEX].rRadius
        p3136911649: stRobotPathPlanner[iRobotSel].stRobotPoints[INDEX].rEndHeight
        p797552052: stRobotPathPlanner[iRobotSel].stRobotPoints[INDEX].bMoveToDone
        p1757482276: Slope Type
        p4236254150: StartHeight
        p580417189: stRobotPathPlanner[iRobotSel].stRobotPoints[INDEX].rStartHeight
        p1744040210: MaxHeight
        p1207913955: stRobotPathPlanner[iRobotSel].stRobotPoints[INDEX].rMaxHeight
    Button (725,382 98x24), "Teach In Point"
        tap stRobotPathPlanner[iRobotSel].stTeachInPoints.bExTeachIn
    Textfield (568,383 142x26), "%s", text variable: stRobotPathPlanner[iRobotSel].stTeachInPoints.usiTeachInPoint
    Textfield (408,386 142x24), "%s", text variable: stRobotPathPlanner[iRobotSel].stTeachInPoints.usiSetPointNo
        OnMouseClick: write the text variable via Default
    Label (408,366 122x14), "Set Teach In Point"
    Label (583,366 122x14), "Actual Teach In Point"
    PushSwitch (378,44 47x61), tooltip "Select Bacis Coordinate System", variable: stRobotCmd[iRobotSel].bBasicCoordSystem, behaviour: TOGGLE, style: Switch-PushSwitch-Gray
    PushSwitch (161,246 47x61), tooltip "Clear Error", variable: stRobotCmd[iRobotSel].bClearError, behaviour: TOGGLE, style: Switch-PushSwitch-Gray
    ComboBoxInteger (36,52 73x26), tooltip "Select robot number", variable: iRobotSel
    Label (54,123 92x14), "Enable"
    Label (80,189 92x14), "Emergency Stop"
    Label (212,126 122x14), "Main Contactor"
    Label (46,262 122x14), "Power On"
    Label (215,262 122x14), "Clear Error"
    Label (430,60 199x14), "Select Basic Coordinate System"
    Label (128,56 85x14), "Select Robot"
    Label (1164,59 134x13), "Jog Coordinate"
    Label (786,73 89x13), "Jog plus"
    Label (1001,72 89x13), "Jog minus"
    Label (1084,70 89x13), "Jog plus"
    Label (1304,69 89x13), "Jog minus"
    Textfield (192,171 158x31), "E-Stop Dec.: %s", text variable: stRobotCmd[iRobotSel].rEmergencyStopDec
        OnMouseClick: write the text variable via Default
    Textfield (868,140 144x29), "Jog Joint Vel.: %s", text variable: stRobotCmd[iRobotSel].stJogJoint.rJogVel
        OnMouseClick: write the text variable via Default
    Textfield (870,176 144x28), "Jog Joint Acc.: %s", text variable: stRobotCmd[iRobotSel].stJogJoint.rJogAcc
        OnMouseClick: write the text variable via Default
    Textfield (870,211 144x28), "Jog Joint Jerk : %s", text variable: stRobotCmd[iRobotSel].stJogJoint.rJogJerk
        OnMouseClick: write the text variable via Default
    Textfield (1163,138 144x29), "Jog Coord.Vel.: %s", text variable: stRobotCmd[iRobotSel].stJogCoordinate.rJogVel
        OnMouseClick: write the text variable via Default
    Textfield (1165,174 144x28), "Jog Coord.Acc.: %s", text variable: stRobotCmd[iRobotSel].stJogCoordinate.rJogAcc
        OnMouseClick: write the text variable via Default
    Textfield (1165,209 144x28), "Jog Coord. Jerk : %s", text variable: stRobotCmd[iRobotSel].stJogCoordinate.rJogJerk
        OnMouseClick: write the text variable via Default
    Textfield (191,206 159x31), "E-Stop Jerk: %s", text variable: stRobotCmd[iRobotSel].rEmergencyStopJerk
        OnMouseClick: write the text variable via Default
    Textfield (849,382 142x24), "%s", text variable: stRobotPathPlanner[iRobotSel].stTeachInPoints.strRecipeFile
        OnMouseClick: write the text variable via Default
    Label (849,357 122x14), "Recipe File Name"
    Button (1142,379 106x24), "Start Command"
        toggle stRobotPathPlanner[iRobotSel].stTeachInPoints.bExRecipeCommand
    Textfield (998,379 130x26), "%s", text variable: stRobotPathPlanner[iRobotSel].stTeachInPoints.enRecipeCommand
        OnMouseClick: write the text variable via Default
    Label (994,358 122x14), "Recipe Command"
    Lamp1 (1269,377 28x36), variable: stRobotPathPlanner[iRobotSel].stTeachInPoints.bRecipeCommandDone, style: Lamp-Lamp1-Green
    Label (1246,356 76x14), "Cmd Done"
    Table (589,104 189x196), data array: stRobotFbk[iRobotSel].arJointCoordinates
        p3854506369: stRobotFbk[iRobotSel].arJointCoordinates[INDEX]
        p1014161805: 16 - 1 + 1
    Lamp1 (38,380 27x36), variable: stRobotFbk[iRobotSel].bAxisPowerOk, style: Lamp-Lamp1-Green
    Lamp1 (108,380 27x36), variable: stRobotFbk[iRobotSel].bAxisHomed, style: Lamp-Lamp1-Green
    Label (78,360 83x14), "Axis Homed"
    Lamp1 (180,379 27x36), variable: stRobotFbk[iRobotSel].bAxisError, style: Lamp-Lamp1-Red
    Label (150,359 83x14), "Axis Error"
    Lamp1 (244,378 27x36), variable: stRobotFbk[iRobotSel].bAxisGrouped, style: Lamp-Lamp1-Green
    Label (216,359 83x14), "Axis Group"
    Lamp1 (311,377 27x36), variable: stRobotFbk[iRobotSel].bKinError, style: Lamp-Lamp1-Red
    Label (281,358 83x14), "Kin Error"
    GroupBox (12,343 371x74), "Robot Status"
    Lamp1 (872,310 28x36), variable: stRobotFbk[iRobotSel].bAxisMoving, style: Lamp-Lamp1-Green
    Lamp1 (1158,310 28x36), variable: stRobotFbk[iRobotSel].bKinMoving, style: Lamp-Lamp1-Green
    Textfield (870,245 144x28), "Jog Joint Override : %s", text variable: stRobotCmd[iRobotSel].stJogJoint.rJogOverride
        OnMouseClick: write the text variable via Default
    Checkbox (867,279 192x30), "Reduce 1/100 jog override", variable: stRobotCmd[iRobotSel].stJogJoint.bCutJogOverrideBy100
    Textfield (1166,242 144x28), "Jog Coord. Override : %s", text variable: stRobotCmd[iRobotSel].stJogCoordinate.rJogOverride
        OnMouseClick: write the text variable via Default
    Checkbox (1163,276 196x30), "Reduce 1/100 jog override", variable: stRobotCmd[iRobotSel].stJogCoordinate.bCutJogOverrideBy100
    Label (910,318 122x14), "Robot Axis Moving"
    Label (1196,318 122x14), "Robot Kin Moving"
    Button (705,341 143x24), "Teach In Aux Circ Point"
        tap stRobotPathPlanner[iRobotSel].stTeachInPoints.bExTeachInAuxCirc
    Label (7,361 83x14), "Axis Power"
    PushSwitch (213,1035 47x61), tooltip "Start Cycle", variable: stRobotPathPlanner[iRobotSel].stPathPlannerCmd.bRunPathPlanner, behaviour: TOGGLE, style: Switch-PushSwitch-Gray
    Label (240,1050 122x14), "Start Cycle"
    Lamp1 (626,960 28x36), variable: stPathPlannerFbk[iRobotSel].bPathCycleActive, style: Lamp-Lamp1-Green
    Label (664,968 122x14), "Path Cycle Active"
    Lamp1 (626,996 28x36), variable: stPathPlannerFbk[iRobotSel].bPathMoveToDone, style: Lamp-Lamp1-Green
    Label (671,1000 122x14), "Path Move To Done"
    Textfield (217,956 130x24), "%s", text variable: stPathPlannerFbk[iRobotSel].usiBufferedBlock
        OnMouseClick: write the text variable via Default
    Label (388,962 149x14), "Path Last Buffered Point"
    PushSwitch (212,1126 47x61), tooltip "Start Cycle", variable: stRobotPathPlanner[iRobotSel].stPathPlannerCmd.bHoldCycle, behaviour: TOGGLE, style: Switch-PushSwitch-Gray
    Label (239,1143 122x14), "Hold Cycle"
    Lamp1 (626,1031 28x36), variable: stPathPlannerFbk[iRobotSel].bHoldCycleActive, style: Lamp-Lamp1-YELLOW
    Label (662,1038 122x14), "Path Hold Active"
    Textfield (49,676 71x23), "%s", text variable: stRobotPathPlanner[iRobotSel].stRobotPoints[iRowSel].strPointName
        OnMouseClick: write the text variable via Default
    Textfield (124,676 88x24), "%s", text variable: stRobotPathPlanner[iRobotSel].stRobotPoints[iRowSel].bEnableCondition
        OnMouseClick: write the text variable via Default
    Textfield (216,676 67x24), "%s", text variable: stRobotPathPlanner[iRobotSel].stRobotPoints[iRowSel].usiJumpBefore
        OnMouseClick: write the text variable via Default
    Textfield (286,676 59x24), "%s", text variable: stRobotPathPlanner[iRobotSel].stRobotPoints[iRowSel].usiJumpAfter
        OnMouseClick: write the text variable via Default
    Textfield (348,676 136x24), "%s", text variable: stRobotPathPlanner[iRobotSel].stRobotPoints[iRowSel].enMotionType
        OnMouseClick: write the text variable via Default
    Textfield (488,676 177x24), "%s", text variable: stRobotPathPlanner[iRobotSel].stRobotPoints[iRowSel].enCoordSys
        OnMouseClick: write the text variable via Default
    Textfield (670,676 171x24), "%s", text variable: stRobotPathPlanner[iRobotSel].stRobotPoints[iRowSel].enSlopeType
        OnMouseClick: write the text variable via Default
    Textfield (848,675 59x24), "%s", text variable: stRobotPathPlanner[iRobotSel].stRobotPoints[iRowSel].enSetMode
        OnMouseClick: write the text variable via Default
    Textfield (910,675 56x24), "%s", text variable: stRobotPathPlanner[iRobotSel].stRobotPoints[iRowSel].rVel
        OnMouseClick: write the text variable via Default
    Textfield (970,675 58x24), "%s", text variable: stRobotPathPlanner[iRobotSel].stRobotPoints[iRowSel].rAcc
        OnMouseClick: write the text variable via Default
    Textfield (1030,675 58x24), "%s", text variable: stRobotPathPlanner[iRobotSel].stRobotPoints[iRowSel].rJerk
        OnMouseClick: write the text variable via Default
    Textfield (1091,674 58x24), "%s", text variable: stRobotPathPlanner[iRobotSel].stRobotPoints[iRowSel].rRadius
        OnMouseClick: write the text variable via Default
    Textfield (1152,674 64x24), "%s", text variable: stRobotPathPlanner[iRobotSel].stRobotPoints[iRowSel].rStartHeight
        OnMouseClick: write the text variable via Default
    Textfield (1222,673 65x24), "%s", text variable: stRobotPathPlanner[iRobotSel].stRobotPoints[iRowSel].rMaxHeight
        OnMouseClick: write the text variable via Default
    Textfield (1290,672 65x24), "%s", text variable: stRobotPathPlanner[iRobotSel].stRobotPoints[iRowSel].rEndHeight
        OnMouseClick: write the text variable via Default
    GroupBox (20,653 1357x279), "End Point Coordinates"
        Button (21,54 98x24), "Delete Block"
            tap stRobotPathPlanner[iRobotSel].stPathPlannerCmd.bDeleteBlock
        Button (22,84 98x24), "Insert Block"
            tap stRobotPathPlanner[iRobotSel].stPathPlannerCmd.bInsertEmptyBlock
        Label (22,188 55x11), "Coord.1"
        Textfield (94,155 73x27), "%s", text variable: stRobotPathPlanner[iRobotSel].stRobotPoints[iRowSel].arPos[2]
            OnMouseClick: write the text variable via Default
        Label (99,188 55x11), "Coord.2"
        Textfield (173,154 73x27), "%s", text variable: stRobotPathPlanner[iRobotSel].stRobotPoints[iRowSel].arPos[3]
            OnMouseClick: write the text variable via Default
        Label (178,187 55x11), "Coord.3"
        Textfield (252,154 73x27), "%s", text variable: stRobotPathPlanner[iRobotSel].stRobotPoints[iRowSel].arPos[4]
            OnMouseClick: write the text variable via Default
        Textfield (331,154 73x27), "%s", text variable: stRobotPathPlanner[iRobotSel].stRobotPoints[iRowSel].arPos[5]
            OnMouseClick: write the text variable via Default
        Textfield (410,154 73x27), "%s", text variable: stRobotPathPlanner[iRobotSel].stRobotPoints[iRowSel].arPos[6]
            OnMouseClick: write the text variable via Default
        Textfield (491,153 73x27), "%s", text variable: stRobotPathPlanner[iRobotSel].stRobotPoints[iRowSel].arPos[7]
            OnMouseClick: write the text variable via Default
        Textfield (570,152 73x27), "%s", text variable: stRobotPathPlanner[iRobotSel].stRobotPoints[iRowSel].arPos[8]
            OnMouseClick: write the text variable via Default
        Label (256,187 55x11), "Coord.4"
        Label (335,187 55x11), "Coord.5"
        Label (418,186 55x10), "Coord.6"
        Label (501,185 55x11), "Coord.7"
        Label (578,184 55x11), "Coord.8"
        Textfield (697,153 73x27), "%s", text variable: stRobotPathPlanner[iRobotSel].stRobotPoints[iRowSel].arAuxPos[1]
            OnMouseClick: write the text variable via Default
        Label (702,186 55x11), "Coord.1"
        Textfield (774,153 73x27), "%s", text variable: stRobotPathPlanner[iRobotSel].stRobotPoints[iRowSel].arAuxPos[2]
            OnMouseClick: write the text variable via Default
        Label (779,186 55x11), "Coord.2"
        Textfield (853,152 73x27), "%s", text variable: stRobotPathPlanner[iRobotSel].stRobotPoints[iRowSel].arAuxPos[3]
            OnMouseClick: write the text variable via Default
        Label (858,185 55x11), "Coord.3"
        Textfield (932,152 73x27), "%s", text variable: stRobotPathPlanner[iRobotSel].stRobotPoints[iRowSel].arAuxPos[4]
            OnMouseClick: write the text variable via Default
        Textfield (1011,152 73x27), "%s", text variable: stRobotPathPlanner[iRobotSel].stRobotPoints[iRowSel].arAuxPos[5]
            OnMouseClick: write the text variable via Default
        Textfield (1090,152 73x27), "%s", text variable: stRobotPathPlanner[iRobotSel].stRobotPoints[iRowSel].arAuxPos[6]
            OnMouseClick: write the text variable via Default
        Textfield (1171,151 73x27), "%s", text variable: stRobotPathPlanner[iRobotSel].stRobotPoints[iRowSel].arAuxPos[7]
            OnMouseClick: write the text variable via Default
        Textfield (1250,150 73x27), "%s", text variable: stRobotPathPlanner[iRobotSel].stRobotPoints[iRowSel].arAuxPos[8]
            OnMouseClick: write the text variable via Default
        Label (936,185 55x11), "Coord.4"
        Label (1015,185 55x11), "Coord.5"
        Label (1098,184 55x10), "Coord.6"
        Label (1181,183 55x11), "Coord.7"
        Label (1258,182 55x11), "Coord.8"
        GroupBox (10,202 646x67), "Belt Values for Syncnronization"
        Textfield (160,55 40x55), "%s", text variable: iCopyBlock
            OnMouseClick: write the text variable via Default
        Button (203,55 98x24), "Copy to Block"
            tap stRobotPathPlanner[iRobotSel].stPathPlannerCmd.bCopyBlock
        Button (205,86 98x24), "Move to Block"
            tap stRobotPathPlanner[iRobotSel].stPathPlannerCmd.bMoveBlock
        Textfield (892,92 56x24), "%s", text variable: stRobotPathPlanner[iRobotSel].stPathPlannerCmd.rPathVelAll
            OnMouseClick: write the text variable via Default
        Textfield (17,156 73x27), "%s", text variable: stRobotPathPlanner[iRobotSel].stRobotPoints[iRowSel].arPos[1]
            OnMouseClick: write the text variable via Default
        GroupBox (687,135 646x67), "Move Circular Intermediate Point Coordinates"
        Textfield (873,250 88x24), "%s", text variable: stRobotPathPlanner[iRobotSel].stMoveCircAddData[iRowSel].bCW_CCW
            OnMouseClick: write the text variable via Default
        Textfield (873,219 177x24), "%s", text variable: stRobotPathPlanner[iRobotSel].stMoveCircAddData[iRowSel].enKinPlane
            OnMouseClick: write the text variable via Default
        Label (690,256 143x14), "Move Circular CW/CCW:"
        Label (689,222 176x14), "Move Circular Plane Selection:"
        Label (960,255 338x14), "( Valid only for 2D plane selection XY,XZ,YZ : False = CW )"
        Textfield (19,220 73x27), "%s", text variable: stRobotPathPlanner[iRobotSel].stRobotPoints[iRowSel].arPos[9]
            OnMouseClick: write the text variable via Default
        GroupBox (10,135 646x67), "End Point Coordinates"
    Textfield (488,715 177x24), "%s", text variable: stRobotPathPlanner[iRobotSel].stPathPlannerCmd.enCoordSysAll
        OnMouseClick: write the text variable via Default
    Textfield (671,715 171x24), "%s", text variable: stRobotPathPlanner[iRobotSel].stPathPlannerCmd.enSlopeAll
        OnMouseClick: write the text variable via Default
    Textfield (849,714 59x24), "%s", text variable: stRobotPathPlanner[iRobotSel].stPathPlannerCmd.enSetModeAll
        OnMouseClick: write the text variable via Default
    Textfield (911,714 56x24), "%s", text variable: stRobotPathPlanner[iRobotSel].stPathPlannerCmd.rPathVelAll
        OnMouseClick: write the text variable via Default
    Textfield (971,714 58x24), "%s", text variable: stRobotPathPlanner[iRobotSel].stPathPlannerCmd.rPathAccAll
        OnMouseClick: write the text variable via Default
    Textfield (1031,714 58x24), "%s", text variable: stRobotPathPlanner[iRobotSel].stPathPlannerCmd.rPathJerkAll
        OnMouseClick: write the text variable via Default
    Textfield (1092,713 58x24), "%s", text variable: stRobotPathPlanner[iRobotSel].stPathPlannerCmd.rPathBlendAll
        OnMouseClick: write the text variable via Default
    Button (1160,711 98x24), "Set All Point Data"
        tap stRobotPathPlanner[iRobotSel].stPathPlannerCmd.bSetPathParAll
    Textfield (972,746 58x24), "%s", text variable: stRobotPathPlanner[iRobotSel].stPathPlannerCmd.rPathAccAll
        OnMouseClick: write the text variable via Default
    Textfield (1032,746 58x24), "%s", text variable: stRobotPathPlanner[iRobotSel].stPathPlannerCmd.rPathJerkAll
        OnMouseClick: write the text variable via Default
    Textfield (1093,745 58x24), "%s", text variable: stRobotPathPlanner[iRobotSel].stPathPlannerCmd.rPathBlendAll
        OnMouseClick: write the text variable via Default
    Button (1161,743 113x24), "Set Dynamic Data"
        tap stRobotPathPlanner[iRobotSel].stPathPlannerCmd.bSetPathDynParAll
    Table (40,956 141x223), data array: stPathPlannerFbk[iRobotSel].arBufferSequence
        p3854506369: stPathPlannerFbk[iRobotSel].arBufferSequence[INDEX]
    GroupBox (18,938 1361x247), "Robot Cycle"
        Lamp1 (883,-624 28x36), variable: stRobotFbk[iRobotSel].bAxisMoving, style: Lamp-Lamp1-Green
        Lamp1 (1169,-624 28x36), variable: stRobotFbk[iRobotSel].bKinMoving, style: Lamp-Lamp1-Green
    Textfield (218,997 127x24), "%s", text variable: stRobotPathPlanner[iRobotSel].stPathPlannerCmd.rSetSpeedOverride
        OnMouseClick: write the text variable via Default
    Label (376,999 149x14), "Speed Override (%)"
    PushSwitch (396,1036 45x53), tooltip "Start Cycle", variable: stRobotPathPlanner[iRobotSel].stPathPlannerCmd.bInTouchProbeStop, behaviour: TOGGLE, style: Switch-PushSwitch-Gray
    Label (437,1055 122x14), "Touch probe stop"
    Textfield (395,1089 173x27), "Probe Stop Dec.: %s", text variable: stRobotPathPlanner[iRobotSel].stPathPlannerCmd.rTouchProbeStopDec
        OnMouseClick: write the text variable via Default
    Textfield (394,1124 174x28), "Probe Stop Jerk: %s", text variable: stRobotPathPlanner[iRobotSel].stPathPlannerCmd.rTouchProbeStopJerk
        OnMouseClick: write the text variable via Default
    Lamp1 (626,1066 28x36), variable: stRobotFbk[iRobotSel].bKinMoving, style: Lamp-Lamp1-Green
    Label (664,1074 122x14), "Robot Kin Moving"
    Lamp1 (626,1102 28x36), variable: stRobotFbk[iRobotSel].bKinStandstill, style: Lamp-Lamp1-Green
    Label (664,1110 122x14), "Robot Kin Stanstill"
    Lamp1 (827,960 28x36), variable: stRobotFbk[iRobotSel].bAxisMoving, style: Lamp-Lamp1-Green
    Label (865,968 122x14), "Robot Axis Moving"
    Lamp1 (827,998 28x36), variable: stRobotFbk[iRobotSel].bAxisStandstill, style: Lamp-Lamp1-Green
    Label (874,1004 122x14), "Robot Axis Standstill"
    Textfield (219,1090 127x24), "Start Block: %s", text variable: stRobotPathPlanner[iRobotSel].stPathPlannerCmd.iStartBlock
        OnMouseClick: write the text variable via Default
    Lamp1 (28,1219 32x32), variable: prgRobotManagement.fbRobotBase[iRobotSel].O_bErrorFB, style: Lamp-Lamp1-Yellow
    Textfield (66,1224 437x26), "%s", text variable: prgRobotManagement.fbRobotBase[iRobotSel].O_strErrorIdent
    Label (507,1229 239x14), "FB Robot Base Management Status"
    Lamp1 (28,1261 32x32), variable: prgRobotManagement.fbRobotPathPlanner[iRobotSel].O_Error, style: Lamp-Lamp1-Yellow
    Textfield (66,1266 437x26), "%s", text variable: stPathPlannerFbk[iRobotSel].strStatusMessage
    Label (529,1272 239x14), "FB Robot Path Planner Management Status"
    Lamp1 (28,1302 32x32), variable: prgRobotManagement.fbRecipeManagement[iRobotSel].O_bError, style: Lamp-Lamp1-Yellow
    Textfield (66,1307 437x26), "%s", text variable: prgRobotManagement.fbRecipeManagement[iRobotSel].O_strErrorIdent
    Label (516,1313 239x14), "FB Robot Recipes Management Status"
    GroupBox (17,1199 771x163), "Robot FB Status"
    DipSwitch (842,30 130x41), tooltip "Enable Jog Joint", variable: stRobotCmd[iRobotSel].stJogJoint.bEnableJogJoint, behaviour: TOGGLE, style: Switch-DipSwitch-Gray
    Label (883,41 134x13), "Enable Jog Joint Axis"
    Label (44,905 55x11), "Coord.9"
    Textfield (116,872 73x27), "%s", text variable: stRobotPathPlanner[iRobotSel].stRobotPoints[iRowSel].arPos[10]
        OnMouseClick: write the text variable via Default
    Label (121,905 55x11), "Coord.10"
    Textfield (195,871 73x27), "%s", text variable: stRobotPathPlanner[iRobotSel].stRobotPoints[iRowSel].arPos[11]
        OnMouseClick: write the text variable via Default
    Label (200,904 55x12), "Coord.11"
    Textfield (274,871 73x27), "%s", text variable: stRobotPathPlanner[iRobotSel].stRobotPoints[iRowSel].arPos[12]
        OnMouseClick: write the text variable via Default
    Textfield (353,871 73x27), "%s", text variable: stRobotPathPlanner[iRobotSel].stRobotPoints[iRowSel].arPos[13]
        OnMouseClick: write the text variable via Default
    Textfield (432,871 73x27), "%s", text variable: stRobotPathPlanner[iRobotSel].stRobotPoints[iRowSel].arPos[14]
        OnMouseClick: write the text variable via Default
    Textfield (513,870 73x27), "%s", text variable: stRobotPathPlanner[iRobotSel].stRobotPoints[iRowSel].arPos[15]
        OnMouseClick: write the text variable via Default
    Textfield (592,869 73x27), "%s", text variable: stRobotPathPlanner[iRobotSel].stRobotPoints[iRowSel].arPos[16]
        OnMouseClick: write the text variable via Default
    Label (278,904 55x11), "Coord.12"
    Label (357,904 55x11), "Coord.13"
    Label (440,903 55x10), "Coord.14"
    Label (523,902 55x11), "Coord.15"
    Label (600,901 55x11), "Coord.16"
    Textfield (398,305 177x24), "%s", text variable: stRobotCmd[iRobotSel].enCoordSystemFbk
        OnMouseClick: write the text variable via Default
END_VISUALIZATION
